// TIA Portal V17 export
// export: Created 2024-09-02T12:50:25.6203118Z, ExportSetting WithDefaults, DisplayName Totally Integrated Automation Portal, DisplayVersion V17, DisplayName TIA Portal Openness, DisplayVersion V17, DisplayName TIA Portal Version Control Interface, DisplayVersion V17, DisplayName STEP 7 Professional, DisplayVersion V17, DisplayName STEP 7 Safety, DisplayVersion V17, DisplayName WinCC Professional, DisplayVersion V17
VAR_GLOBAL   // PLC tag table "Camera"
   PLC_Out_For_Omron AT %Q4000.0 : "Omron_PLC_Output_O";
   PLC_Input_Form_Omron AT %I4000.0 : "Omron_PLC_Input_O";
   IBN0MES AT %M2.0 : Bool;
   MessBypased AT %M2.1 : Bool;
   Isynchro1 AT %M2.2 : Bool;
   Isynchro2 AT %M2.3 : Bool;
   Isynchro3 AT %M2.4 : Bool;
   mTempMESPOPUP_EKSBYPASS AT %M500.1 : Bool;
   test_amister AT %M666.0 : Bool;
END_VAR
VAR_GLOBAL CONSTANT   // user constants
   Camera_OK : DWord := 1;
   Camera_NOK : DWord := -1;
END_VAR
